(* IEC 61131-3 sources: SRCI/RobotLibrary/Library/POUs/General/MC_RobotTask (part 3) *)

           // Create log entry
           CreateLogMessagePara3 ( Timestamp   := SystemTime,
                                   MessageType := MessageType.CMD,
                                   Severity    := Severity.DEBUG,
                                   MessageCode := 0,
                                   MessageText := 'SyncLoadData: Synchronization of Load[{1}] triggered by PLC, SyncMode = {2}, SyncTime = {3}, SyncDirection = PLC -> RC',
                                   Para1       :=  DINT_TO_STRING(_rSyncIdx),
                                   Para2       :=  SYNC_MODE_TO_STRING(AxesGroup.Parameter.Plc.Parameter.SynchronizationModes.Load[SyncTime.AFTER_START_UP]),
                                   Para3       :=  SYNC_TIME_TO_STRING(SyncTime.AFTER_START_UP));
                                   RETURN;
         END_IF

         // Conflict triggered by RC ?
         IF ( NOT AxesGroup.State.SyncStateRc.InSync.Load )
         THEN
           // get changed index
          _rSyncIdx := LIMIT(1, AxesGroup.State.SyncStateRc.UnSyncNo.Load, AxesGroup.State.UnifiedLoadIndex); //  !!! Attention : 0 is not allowed - LoadData starts with 1 !!!
           // set timeout
           SetTimeout(PT := _rTimeout, rTimer := _rTimer);
           // inc step counter
          _rStep := 20; // -> read RC data an write it to PLC

           // Create log entry
           CreateLogMessagePara3 ( Timestamp   := SystemTime,
                                   MessageType := MessageType.CMD,
                                   Severity    := Severity.DEBUG,
                                   MessageCode := 0,
                                   MessageText := 'SyncLoadData: Synchronization of Load[{1}] triggered by RC, SyncMode = {2}, SyncTime = {3}, SyncDirection = RC -> PLC',
                                   Para1       :=  DINT_TO_STRING(_rSyncIdx),
                                   Para2       :=  SYNC_MODE_TO_STRING(AxesGroup.Parameter.Plc.Parameter.SynchronizationModes.Load[SyncTime.AFTER_START_UP]),
                                   Para3       :=  SYNC_TIME_TO_STRING(SyncTime.AFTER_START_UP));
                                   RETURN;
  			 END_IF

         // set timeout
         SetTimeout(PT := _rTimeout, rTimer := _rTimer);
         // jump back
        //_rStep := 10;

    // ------------------------------------------
    // Read Data from RC and write it to PLC
    // ------------------------------------------
    20 : IF (( NOT _readLoadData.Busy  ) AND
             ( NOT _readLoadData.Error ))
         THEN
           // set command parameter
          _readLoadData.ParCmd.LoadNo := _rSyncIdx;
           // execute command
          _readLoadData.Execute := TRUE;
           // set timeout
           SetTimeout(PT := _rTimeout, rTimer := _rTimer);
           // inc step counter
          _rStep := _rStep + 1;
         ELSE
           // check error ?
           IF (_readLoadData.Error)
           THEN
             ErrorID     := _readLoadData.ErrorID;
             ErrorAddTxt := _readLoadData.ErrorAddTxt;
           END_IF

           // timeout exceeded ?
           IF (CheckTimeout(_rTimer) = RobotLibraryConstants.OK)
           THEN
             ErrorID     := RobotLibraryErrorIdEnum.ERR_TIMEOUT_CMD;
             ErrorAddTxt := CONCAT(_stepName, DINT_TO_STRING(_rStep));
           END_IF
         END_IF

    21 : IF (( NOT _readLoadData.Busy  ) AND
             ( NOT _readLoadData.Error ) AND
             (     _readLoadData.Done  ))
         THEN
           // reset execution
          _readLoadData.Execute := FALSE;
           // update internal Load data
           LoadData[_rSyncIdx].Data := _readLoadData.OutCmd.LoadData;
          _loadData[_rSyncIdx].Data := _readLoadData.OutCmd.LoadData;
           // set available bit
           LoadData[_rSyncIdx].Available := TRUE;
          _loadData[_rSyncIdx].Available := TRUE;
           // set timeout
           SetTimeout(PT := _rTimeout, rTimer := _rTimer);
           // inc step counter
          _rStep := 10; // -> jump to after startup
         ELSE
           // check error ?
           IF (_readLoadData.Error)
           THEN
             ErrorID     := _readLoadData.ErrorID;
             ErrorAddTxt := _readLoadData.ErrorAddTxt;
             // reset available bit
             LoadData[_rSyncIdx].Available := FALSE;
            _loadData[_rSyncIdx].Available := FALSE;
           END_IF

           // timeout exceeded ?
           IF (CheckTimeout(_rTimer) = RobotLibraryConstants.OK)
           THEN
             ErrorID     := RobotLibraryErrorIdEnum.ERR_TIMEOUT_CMD;
             ErrorAddTxt := CONCAT(_stepName, DINT_TO_STRING(_rStep));
           END_IF
         END_IF

    // ------------------------------------------
    // Write data from PLC to RC
    // ------------------------------------------
    30 : IF (( NOT _writeLoadData.Busy  ) AND
             ( NOT _writeLoadData.Error ))
         THEN
           // set command parameter
          _writeLoadData.ParCmd.LoadNo   := _rSyncIdx;
          _writeLoadData.ParCmd.LoadData :=  LoadData[_rSyncIdx].Data;
           // execute command
          _writeLoadData.Execute := TRUE;
           // set timeout
           SetTimeout(PT := _rTimeout, rTimer := _rTimer);
           // inc step counter
          _rStep := _rStep + 1;
         ELSE
           // check error ?
           IF (_writeLoadData.Error)
           THEN
             ErrorID     := _writeLoadData.ErrorID;
             ErrorAddTxt := _writeLoadData.ErrorAddTxt;;
           END_IF

           // timeout exceeded ?
           IF (CheckTimeout(_rTimer) = RobotLibraryConstants.OK)
           THEN
             ErrorID     := RobotLibraryErrorIdEnum.ERR_TIMEOUT_CMD;
             ErrorAddTxt := CONCAT(_stepName, DINT_TO_STRING(_rStep));
           END_IF
         END_IF

    31 : IF (( NOT _writeLoadData.Busy  ) AND
             ( NOT _writeLoadData.Error ) AND
             (     _writeLoadData.Done  ))
         THEN
           // execute command
          _writeLoadData.Execute := FALSE;
           // update internal Load data
          _loadData[_rSyncIdx] := LoadData[_rSyncIdx];
           // set available bit
           LoadData[_rSyncIdx].Available := TRUE;
          _loadData[_rSyncIdx].Available := TRUE;
           // set timeout
           SetTimeout(PT := _rTimeout, rTimer := _rTimer);
           // inc step counter
          _rStep := 10; // -> jump to after startup;
         ELSE
           // check error ?
           IF (_writeLoadData.Error)
           THEN
             WarningID := RobotLibraryWarningIdEnum.WARN_LOAD_SYNC_FAILED_BY_ERROR_OF_READ_OR_WRITE_CMD;
             // reset available bit
             LoadData[_rSyncIdx].Available := FALSE;
            _loadData[_rSyncIdx].Available := FALSE;
           END_IF

           // timeout exceeded ?
           IF (CheckTimeout(_rTimer) = RobotLibraryConstants.OK)
           THEN
             ErrorID     := RobotLibraryErrorIdEnum.ERR_TIMEOUT_CMD;
             ErrorAddTxt := CONCAT(_stepName, DINT_TO_STRING(_rStep));
           END_IF
         END_IF

  ELSE
    // invalid step
    ErrorID     := RobotLibraryErrorIdEnum.ERR_INVALID_STEP;
    ErrorAddTxt := CONCAT(_stepName , DINT_TO_STRING(_stepCmd));
  END_CASE

END_METHOD

METHOD PRIVATE HandleSyncRobotDefaultDynamics
VAR_IN_OUT
   /// Robot assignment of function
  AxesGroup       : AxesGroup;
  /// Default dynamics stored on PLC. For more information refer to 5.5.7
  DefaultDynamics : DefaultDynamics;
END_VAR

VAR
  /// Internal step counter name
 _stepName        : STRING;
  /// Internal reference to step counter
 _rStep           : REFERENCE TO DINT;
  /// Internal reference to timer
 _rTimer          : REFERENCE TO TON;
  /// Internal reference to timeout
 _rTimeout        : REFERENCE TO TIME;
  /// Internal reference to synchroniztion index
 _rSyncIdx        : REFERENCE TO USINT;
  /// internal bit for condition found
 _found           : BOOL;
  /// empty data set to reset all DataChanged bits
 _dataChangedNone : AxesGroupStateDataChanged;
END_VAR

  // Set internal references
  _stepName      :=   '_stepSyncDefaultDynamics = ';
  _rStep       REF=    _stepSyncDefaultDynamics;
  _rTimer      REF=   _timerSyncDefaultDynamics;
  _rTimeout    REF= _timeoutSyncDefaultDynamics;

  CASE _rStep
  OF
    0: // Check initialisation configured ?
       IF (( _parCfg.PLC.Parameter.SynchronizationModes.DefaultDynamics[SyncTime.DURING_START_UP] = SyncMode.NO_SYNCHRONIZATION ) AND
           ( _parCfg.PLC.Parameter.SynchronizationModes.DefaultDynamics[SyncTime. AFTER_START_UP] = SyncMode.NO_SYNCHRONIZATION ))
       THEN
         RETURN;
       END_IF

       // wait for initialisation done
       IF  ((     AxesGroup.State.RobotData.RCSupportedFunctions .ReadRobotDefaultDynamics ) AND
            (     AxesGroup.State.RobotData.RCSupportedFunctions.WriteRobotDefaultDynamics ) AND
            (     AxesGroup.State.Initialized                                              ) AND
            ( NOT Error                                                                    ))
       THEN
         // Create log entry
         CreateLogMessagePara1 ( Timestamp   := SystemTime,
                                 MessageType := MessageType.CMD,
                                 Severity    := Severity.DEBUG,
                                 MessageCode := 0,
                                 MessageText := 'SyncDefaultDynamics: Start initial reading of DefaultDynamics from RC',
                                 Para1       :=  '');

         // set timeout
         SetTimeout(PT := _rTimeout, rTimer := _rTimer);
         // inc step counter
        _rStep := _rStep + 1;
       END_IF

       // Start read DefaultDynamics
    1: IF (( NOT _readRobotDefaultDynamics .Busy  ) AND
           ( NOT _readRobotDefaultDynamics.Error ))
       THEN
         // execute command
        _readRobotDefaultDynamics.Execute := TRUE;
         // set timeout
         SetTimeout(PT := _rTimeout, rTimer := _rTimer);
         // inc step counter
        _rStep := _rStep + 1;
       ELSE
         // check error ?
         IF ( _readRobotDefaultDynamics.Error ) AND ( WarningID = RobotLibraryWarningIdEnum.NO_WARNING )
         THEN
           WarningID := RobotLibraryWarningIdEnum.WARN_DEFAULT_DYNAMICS_SYNC_FAILED_BY_ERROR_OF_READ_OR_WRITE_CMD;
         END_IF

         // timeout exceeded ?
         IF (CheckTimeout(_rTimer) = RobotLibraryConstants.OK)
         THEN
           ErrorID     := RobotLibraryErrorIdEnum.ERR_TIMEOUT_CMD;
           ErrorAddTxt := CONCAT(_stepName, DINT_TO_STRING(_rStep));
         END_IF
       END_IF

       // Wait DefaultDynamics read
    2: IF (( NOT _readRobotDefaultDynamics.Busy  ) AND
           ( NOT _readRobotDefaultDynamics.Error ) AND
           (     _readRobotDefaultDynamics.Done  ))
       THEN
         // reset execution
        _readRobotDefaultDynamics.Execute := FALSE;
         // Copy data
        _defaultDynamics := _readRobotDefaultDynamics.OutCmd.DynamicValues;
         // Set plc in sync flag
         AxesGroup.State.SyncStatePlc.InSync.DefaultDynamics := TRUE;

         // Check DefaultDynamics data is equal ?
         IF ( NOT IsDefaultDynamicsEqual( Data1 := _defaultDynamics, Data2 := DefaultDynamics, IgnoreTimestamp := TRUE))
         THEN
           // Reset plc in sync flag
           AxesGroup.State.SyncStatePlc.InSync.DefaultDynamics := FALSE;
           // Set data changed flag
           AxesGroup.State.DataChanged.DefaultDynamics := TRUE;
           // set timeout
           SetTimeout(PT := _rTimeout, rTimer := _rTimer);
           // inc step counter
          _rStep := _rStep + 1;

           // Create log entry
           CreateLogMessagePara1 ( Timestamp   := SystemTime,
                                   MessageType := MessageType.CMD,
                                   Severity    := Severity.DEBUG,
                                   MessageCode := 0,
                                   MessageText := 'SyncDefaultDynamics: Detected a difference in DefaultDynamics between PLC and RC',
                                   Para1       :=  '');

           // Check synchronisation is enabled ?
           IF ( NOT  AxesGroup.State.DataEnableSync.EnableSyncDefaultDynamics ) AND (InfoID = RobotLibraryInfoIdEnum.NO_INFO )
           THEN
             InfoID := RobotLibraryInfoIdEnum.INFO_SYNC_DEFAULT_DYNAMICS_DISABLED;
  				 END_IF

           // Check user interaction needed ?
           IF ( AxesGroup.Parameter.Plc.Parameter.SyncUserInteraction.DefaultDynamics ) AND ( WarningID = RobotLibraryWarningIdEnum.NO_WARNING )
           THEN
             WarningID := RobotLibraryWarningIdEnum.WARN_DEFAULT_DYNAMICS_SYNC_ERROR;
  				 END_IF
  			 END_IF
       ELSE
         // check error ?
         IF (_readRobotDefaultDynamics.Error)
         THEN
           // Set warning
           WarningID := RobotLibraryWarningIdEnum.WARN_DEFAULT_DYNAMICS_SYNC_FAILED_BY_ERROR_OF_READ_OR_WRITE_CMD;
         END_IF

         // timeout exceeded ?
         IF (CheckTimeout(_rTimer) = RobotLibraryConstants.OK)
         THEN
           ErrorID     := RobotLibraryErrorIdEnum.ERR_TIMEOUT_CMD;
           ErrorAddTxt := CONCAT(_stepName, DINT_TO_STRING(_rStep));
         END_IF
       END_IF

       // Check synchronisation state ?
    3: IF ((  NOT AxesGroup.State.DataChanged.DefaultDynamics                                                                                    ) OR
           (      AxesGroup.Parameter.Plc.Parameter.SynchronizationModes.DefaultDynamics[SyncTime.DURING_START_UP] = SyncMode.NO_SYNCHRONIZATION ))
       THEN
         // Update bit for data in sync
         AxesGroup.State.SyncStatePlc.InSync.DefaultDynamics := NOT AxesGroup.State.DataChanged.DefaultDynamics ;
         // set timeout
         SetTimeout(PT := _rTimeout, rTimer := _rTimer);
         // inc step counter
        _rStep := 10; // -> jump to after startup

         // Create log entry
         CreateLogMessagePara1 ( Timestamp   := SystemTime,
                                 MessageType := MessageType.CMD,
                                 Severity    := Severity.DEBUG,
                                 MessageCode := 0,
                                 MessageText := 'SyncDefaultDynamics: Synchronization Startup Phase done',
                                 Para1       :=  '' );
       ELSE
         // Check user interaction needed ?
         IF ( NOT AxesGroup.Parameter.Plc.Parameter.SyncUserInteraction.DefaultDynamics )
         THEN
           CASE AxesGroup.Parameter.Plc.Parameter.SynchronizationModes.DefaultDynamics[SyncTime.DURING_START_UP] OF

             SyncMode.SERVER_TO_CLIENT :

               // Overwrite PLC data with RC data
               DefaultDynamics := _defaultDynamics;
               // Reset data changed flags
               AxesGroup.State.DataChanged.DefaultDynamics := _dataChangedNone.DefaultDynamics;
               // Reset Synchronizing flag
               AxesGroup.State.Synchronizing.DefaultDynamics := FALSE;
               // Set plc in sync flag
               AxesGroup.State.SyncStatePlc.InSync.DefaultDynamics := TRUE;
               // set timeout
               SetTimeout(PT := _rTimeout, rTimer := _rTimer);
               // inc step counter
              _rStep := 10; // -> jump to after startup

              // Create log entry
              CreateLogMessagePara2 ( Timestamp   := SystemTime,
                                      MessageType := MessageType.CMD,
                                      Severity    := Severity.DEBUG,
                                      MessageCode := 0,
                                      MessageText := 'SyncDefaultDynamics: Synchronization of DefaultDynamics triggered by StartUp-Compare, SyncMode = {1}, SyncTime = {2}, SyncDirection = RC -> PLC',
                                      Para1       :=  SYNC_MODE_TO_STRING(AxesGroup.Parameter.Plc.Parameter.SynchronizationModes.DefaultDynamics[SyncTime.DURING_START_UP]),
                                      Para2       :=  SYNC_TIME_TO_STRING(SyncTime.DURING_START_UP));
              // Create log entry
              CreateLogMessagePara1 ( Timestamp   := SystemTime,
                                      MessageType := MessageType.CMD,
                                      Severity    := Severity.DEBUG,
                                      MessageCode := 0,
                                      MessageText := 'SyncDefaultDynamics: Applied the initial read DefaultDynamics from RC',
                                      Para1       :=  '' );

  				   SyncMode.CLIENT_TO_SERVER : ;

               IF ( AxesGroup.State.DataChanged.DefaultDynamics )
               THEN
                 // Reset plc in sync flag
                 AxesGroup.State.SyncStatePlc.InSync.DefaultDynamics := FALSE;
                 // Set Synchronizing flag
                 AxesGroup.State.Synchronizing.DefaultDynamics := TRUE;
                 // set timeout
                 SetTimeout(PT := _rTimeout, rTimer := _rTimer);
                 // inc step counter
                _rStep := _rStep +1; // -> write PLC data to RC
                 // Create log entry
                 CreateLogMessagePara2 ( Timestamp   := SystemTime,
                                         MessageType := MessageType.CMD,
                                         Severity    := Severity.DEBUG,
                                         MessageCode := 0,
                                         MessageText := 'SyncDefaultDynamics: Synchronization of DefaultDynamics triggered by StartUp-Compare, SyncMode = {1}, SyncTime = {2}, SyncDirection = PLC -> RC',
                                         Para1       :=  SYNC_MODE_TO_STRING(AxesGroup.Parameter.Plc.Parameter.SynchronizationModes.DefaultDynamics[SyncTime.DURING_START_UP]),
                                         Para2       :=  SYNC_TIME_TO_STRING(SyncTime.DURING_START_UP));
               ELSE
                 // Reset data changed flags
                 AxesGroup.State.DataChanged.DefaultDynamics := _dataChangedNone.DefaultDynamics;
                 // Reset Synchronizing flag
                 AxesGroup.State.Synchronizing.DefaultDynamics := FALSE;
                 // Set plc in sync flag
                 AxesGroup.State.SyncStatePlc.InSync.DefaultDynamics := TRUE;
                 // set timeout
                 SetTimeout(PT := _rTimeout, rTimer := _rTimer);
                 // inc step counter
                _rStep := 10; // -> jump to after startup
  				     END_IF
           ELSE
             // invalid sync mode for startup
             ErrorID := RobotLibraryErrorIdEnum.ERR_SYNC_MODE_INVALID;
   	       END_CASE
         END_IF
       END_IF

       // Start write DefaultDynamics data
    4: IF (( NOT _writeRobotDefaultDynamics.Busy  ) AND
           ( NOT _writeRobotDefaultDynamics.Error ))
       THEN
         // set command parameter
        _writeRobotDefaultDynamics.ParCmd.DynamicValues :=  DefaultDynamics;
         // execute command
        _writeRobotDefaultDynamics.Execute := TRUE;
         // set timeout
         SetTimeout(PT := _rTimeout, rTimer := _rTimer);
         // inc step counter
        _rStep := _rStep + 1;
       ELSE
         // check error ?
         IF (_writeRobotDefaultDynamics.Error)
         THEN
           ErrorID     := _writeRobotDefaultDynamics.ErrorID;
           ErrorAddTxt := _writeRobotDefaultDynamics.ErrorAddTxt;;
         END_IF

         // timeout exceeded ?
         IF (CheckTimeout(_rTimer) = RobotLibraryConstants.OK)
         THEN
           ErrorID     := RobotLibraryErrorIdEnum.ERR_TIMEOUT_CMD;
           ErrorAddTxt := CONCAT(_stepName, DINT_TO_STRING(_rStep));
         END_IF
       END_IF

       // Wait DefaultDynamics data written ?
    5: IF (( NOT _writeRobotDefaultDynamics.Busy  ) AND
           ( NOT _writeRobotDefaultDynamics.Error ) AND
           (     _writeRobotDefaultDynamics.Done  ))
       THEN
         // execute command
        _writeRobotDefaultDynamics.Execute := FALSE;
         // apply DefaultDynamics data to internal DefaultDynamics data
        _defaultDynamics := DefaultDynamics;
         // reset data changed bit
         AxesGroup.State.DataChanged.DefaultDynamics := FALSE;
         // set timeout
         SetTimeout(PT := _rTimeout, rTimer := _rTimer);
         // dec step counter
        _rStep := _rStep - 2;
       ELSE
         // check error ?
         IF (_writeRobotDefaultDynamics.Error)
         THEN
           WarningID := RobotLibraryWarningIdEnum.WARN_DEFAULT_DYNAMICS_SYNC_FAILED_BY_ERROR_OF_READ_OR_WRITE_CMD;
         END_IF

         // timeout exceeded ?
         IF (CheckTimeout(_rTimer) = RobotLibraryConstants.OK)
         THEN
           ErrorID     := RobotLibraryErrorIdEnum.ERR_TIMEOUT_CMD;
           ErrorAddTxt := CONCAT(_stepName, DINT_TO_STRING(_rStep));
         END_IF
       END_IF

    // --------------------------------------------
    // SyncMode after startup :
    // --------------------------------------------

    10 :// check synchronisation active ?
         IF ( AxesGroup.Parameter.Plc.Parameter.SynchronizationModes.DefaultDynamics[SyncTime.AFTER_START_UP] = SyncMode.NO_SYNCHRONIZATION)
         THEN
           RETURN;
         END_IF

         // compare DefaultDynamics data
         AxesGroup.State.DataChanged.DefaultDynamics := NOT IsDefaultDynamicsEqual( Data1 := DefaultDynamics, Data2 := _defaultDynamics, IgnoreTimestamp := FALSE);

         // Check DefaultDynamics data changed ?
         IF (AxesGroup.State.DataChanged.DefaultDynamics)
         THEN
           // Create log entry
           CreateLogMessagePara1 ( Timestamp   := SystemTime,
                                   MessageType := MessageType.CMD,
                                   Severity    := Severity.DEBUG,
                                   MessageCode := 0,
                                   MessageText := 'SyncDefaultDynamics: Detected a local change of DefaultDynamics on PLC, SyncTime = {1}',
                                   Para1       :=  SYNC_TIME_TO_STRING(SyncTime.AFTER_START_UP));
         END_IF

         // Update plc in sync flag
         AxesGroup.State.SyncStatePlc.InSync.DefaultDynamics := NOT AxesGroup.State.DataChanged.DefaultDynamics;

         // Check synchronization is needed ?
         IF ( NOT AxesGroup.State.SyncStatePlc.InSync.DefaultDynamics ) XOR
            ( NOT AxesGroup.State.SyncStateRc .InSync.DefaultDynamics )
         THEN
           CASE AxesGroup.Parameter.Plc.Parameter.SynchronizationModes.DefaultDynamics[SyncTime.AFTER_START_UP]
           OF
             // NO_SYNCHRONIZATION
             SyncMode.NO_SYNCHRONIZATION : ; // no further action

             // CLIENT_TO_SERVER
             SyncMode.CLIENT_TO_SERVER :
               // set timeout
               SetTimeout(PT := _rTimeout, rTimer := _rTimer);
               // inc step counter
              _rStep := 11;

             // SERVER_TO_CLIENT
             SyncMode.SERVER_TO_CLIENT :
               // set timeout
               SetTimeout(PT := _rTimeout, rTimer := _rTimer);
               // inc step counter
              _rStep := 12;

             // AUTOMATIC
             SyncMode.AUTOMATIC :
               // set timeout
               SetTimeout(PT := _rTimeout, rTimer := _rTimer);
               // inc step counter
              _rStep := 13;
           END_CASE
         ELSE
           // datas changeḍ on both sides ? -> Warning
           IF (( NOT AxesGroup.State.SyncStatePlc.InSync.DefaultDynamics ) AND
               ( NOT AxesGroup.State.SyncStateRc .InSync.DefaultDynamics ))
           THEN
             WarningID := RobotLibraryWarningIdEnum.WARN_DEFAULT_DYNAMICS_SYNC_BOTH_SIDES_CHANGED;
           END_IF
         END_IF

    // ------------------------------------------
    // SyncMode : CLIENT_TO_SERVER
    // ------------------------------------------
    11 : // Conflict triggerd by PLC ?
         IF ( NOT AxesGroup.State.SyncStatePlc.InSync.DefaultDynamics )
         THEN
           // set timeout
           SetTimeout(PT := _rTimeout, rTimer := _rTimer);
           // inc step counter
          _rStep := 30; // -> write PLC data to RC

           // Create log entry
           CreateLogMessagePara2 ( Timestamp   := SystemTime,
                                   MessageType := MessageType.CMD,
                                   Severity    := Severity.DEBUG,
                                   MessageCode := 0,
                                   MessageText := 'SyncDefaultDynamics: Synchronization of DefaultDynamics triggered by PLC, SyncMode = {1}, SyncTime = {2}, SyncDirection = PLC -> RC',
                                   Para1       :=  SYNC_MODE_TO_STRING(AxesGroup.Parameter.Plc.Parameter.SynchronizationModes.DefaultDynamics[SyncTime.AFTER_START_UP]),
                                   Para2       :=  SYNC_TIME_TO_STRING(SyncTime.AFTER_START_UP));
                                   RETURN;
         END_IF

         // Conflict triggered by RC ?
         IF ( NOT AxesGroup.State.SyncStateRc.InSync.DefaultDynamics )
         THEN
           // set timeout
           SetTimeout(PT := _rTimeout, rTimer := _rTimer);
           // inc step counter
          _rStep := 30; // -> write PLC data to RC

           // Create log entry
           CreateLogMessagePara2 ( Timestamp   := SystemTime,
                                   MessageType := MessageType.CMD,
                                   Severity    := Severity.DEBUG,
                                   MessageCode := 0,
                                   MessageText := 'SyncDefaultDynamics: Synchronization of DefaultDynamics triggered by RC, SyncMode = {1}, SyncTime = {2}, SyncDirection = PLC -> RC',
                                   Para1       :=  SYNC_MODE_TO_STRING(AxesGroup.Parameter.Plc.Parameter.SynchronizationModes.DefaultDynamics[SyncTime.AFTER_START_UP]),
                                   Para2       :=  SYNC_TIME_TO_STRING(SyncTime.AFTER_START_UP));
                                   RETURN;
  			 END_IF

         // set timeout
         SetTimeout(PT := _rTimeout, rTimer := _rTimer);
         // jump back
        _rStep := 10;

    // ------------------------------------------
    // SyncMode : SERVER_TO_CLIENT
    // ------------------------------------------
    12 : // Conflict triggerd by PLC ?
         IF ( NOT AxesGroup.State.SyncStatePlc.InSync.DefaultDynamics )
         THEN
           // set timeout
           SetTimeout(PT := _rTimeout, rTimer := _rTimer);
           // inc step counter
          _rStep := 20; // -> read RC data and write it to PLC

           // Create log entry
           CreateLogMessagePara2 ( Timestamp   := SystemTime,
                                   MessageType := MessageType.CMD,
                                   Severity    := Severity.DEBUG,
                                   MessageCode := 0,
                                   MessageText := 'SyncDefaultDynamics: Synchronization of DefaultDynamics triggered by PLC, SyncMode = {1}, SyncTime = {2}, SyncDirection = RC -> PLC',
                                   Para1       :=  SYNC_MODE_TO_STRING(AxesGroup.Parameter.Plc.Parameter.SynchronizationModes.DefaultDynamics[SyncTime.AFTER_START_UP]),
                                   Para2       :=  SYNC_TIME_TO_STRING(SyncTime.AFTER_START_UP));
                                   RETURN;
         END_IF

         // Conflict triggered by RC ?
         IF ( NOT AxesGroup.State.SyncStateRc.InSync.DefaultDynamics )
         THEN
           // set timeout
           SetTimeout(PT := _rTimeout, rTimer := _rTimer);
           // inc step counter
          _rStep := 20; // -> read RC data and write it to PLC

           // Create log entry
           CreateLogMessagePara2 ( Timestamp   := SystemTime,
                                   MessageType := MessageType.CMD,
                                   Severity    := Severity.DEBUG,
                                   MessageCode := 0,
                                   MessageText := 'SyncDefaultDynamics: Synchronization of DefaultDynamics triggered by RC, SyncMode = {1}, SyncTime = {2}, SyncDirection = RC -> PLC',
                                   Para1       :=  SYNC_MODE_TO_STRING(AxesGroup.Parameter.Plc.Parameter.SynchronizationModes.DefaultDynamics[SyncTime.AFTER_START_UP]),
                                   Para2       :=  SYNC_TIME_TO_STRING(SyncTime.AFTER_START_UP));
                                   RETURN;
  			 END_IF

         // set timeout
         SetTimeout(PT := _rTimeout, rTimer := _rTimer);
         // jump back
        _rStep := 10;

    // ------------------------------------------
    // SyncMode : AUTOMATIC
    // ------------------------------------------
    13 : // Conflict triggerd by PLC ?
         IF ( NOT AxesGroup.State.SyncStatePlc.InSync.DefaultDynamics )
         THEN
           // set timeout
           SetTimeout(PT := _rTimeout, rTimer := _rTimer);
           // inc step counter
          _rStep := 30; // -> write PLC data to RC

           // Create log entry
           CreateLogMessagePara2 ( Timestamp   := SystemTime,
                                   MessageType := MessageType.CMD,
                                   Severity    := Severity.DEBUG,
                                   MessageCode := 0,
                                   MessageText := 'SyncDefaultDynamics: Synchronization of DefaultDynamics triggered by PLC, SyncMode = {1}, SyncTime = {2}, SyncDirection = PLC -> RC',
                                   Para1       :=  SYNC_MODE_TO_STRING(AxesGroup.Parameter.Plc.Parameter.SynchronizationModes.DefaultDynamics[SyncTime.AFTER_START_UP]),
                                   Para2       :=  SYNC_TIME_TO_STRING(SyncTime.AFTER_START_UP));
                                   RETURN;
         END_IF

         // Conflict triggered by RC ?
         IF ( NOT AxesGroup.State.SyncStateRc.InSync.DefaultDynamics )
         THEN
           // set timeout
           SetTimeout(PT := _rTimeout, rTimer := _rTimer);
           // inc step counter
          _rStep := 20; // -> read RC data an write it to PLC

           // Create log entry
           CreateLogMessagePara2 ( Timestamp   := SystemTime,
                                   MessageType := MessageType.CMD,
                                   Severity    := Severity.DEBUG,
                                   MessageCode := 0,
                                   MessageText := 'SyncDefaultDynamics: Synchronization of DefaultDynamics triggered by RC, SyncMode = {1}, SyncTime = {2}, SyncDirection = RC -> PLC',
                                   Para1       :=  SYNC_MODE_TO_STRING(AxesGroup.Parameter.Plc.Parameter.SynchronizationModes.DefaultDynamics[SyncTime.AFTER_START_UP]),
                                   Para2       :=  SYNC_TIME_TO_STRING(SyncTime.AFTER_START_UP));
                                   RETURN;
  			 END_IF

         // set timeout
         SetTimeout(PT := _rTimeout, rTimer := _rTimer);
         // jump back
        //_rStep := 10;

    // ------------------------------------------
    // Read Data from RC and write it to PLC
    // ------------------------------------------
    20 : IF (( NOT _readRobotDefaultDynamics.Busy  ) AND
             ( NOT _readRobotDefaultDynamics.Error ))
         THEN
           // execute command
          _readRobotDefaultDynamics.Execute := TRUE;
           // set timeout
           SetTimeout(PT := _rTimeout, rTimer := _rTimer);
           // inc step counter
          _rStep := _rStep + 1;
         ELSE
           // check error ?
           IF (_readRobotDefaultDynamics.Error)
           THEN
             ErrorID     := _readRobotDefaultDynamics.ErrorID;
             ErrorAddTxt := _readRobotDefaultDynamics.ErrorAddTxt;
           END_IF

           // timeout exceeded ?
           IF (CheckTimeout(_rTimer) = RobotLibraryConstants.OK)
           THEN
             ErrorID     := RobotLibraryErrorIdEnum.ERR_TIMEOUT_CMD;
             ErrorAddTxt := CONCAT(_stepName, DINT_TO_STRING(_rStep));
           END_IF
         END_IF

    21 : IF (( NOT _readRobotDefaultDynamics.Busy  ) AND
             ( NOT _readRobotDefaultDynamics.Error ) AND
             (     _readRobotDefaultDynamics.Done  ))
         THEN
           // reset execution
          _readRobotDefaultDynamics.Execute := FALSE;
           // update internal DefaultDynamics data
           DefaultDynamics := _readRobotDefaultDynamics.OutCmd.DynamicValues;
          _defaultDynamics := _readRobotDefaultDynamics.OutCmd.DynamicValues;
           // set timeout
           SetTimeout(PT := _rTimeout, rTimer := _rTimer);
           // inc step counter
          _rStep := 10; // -> jump to after startup
         ELSE
           // check error ?
           IF (_readRobotDefaultDynamics.Error)
           THEN
             ErrorID     := _readRobotDefaultDynamics.ErrorID;
             ErrorAddTxt := _readRobotDefaultDynamics.ErrorAddTxt;
           END_IF

           // timeout exceeded ?
           IF (CheckTimeout(_rTimer) = RobotLibraryConstants.OK)
           THEN
             ErrorID     := RobotLibraryErrorIdEnum.ERR_TIMEOUT_CMD;
             ErrorAddTxt := CONCAT(_stepName, DINT_TO_STRING(_rStep));
           END_IF
         END_IF

    // ------------------------------------------
    // Write data from PLC to RC
    // ------------------------------------------
    30 : IF (( NOT _writeRobotDefaultDynamics.Busy  ) AND
             ( NOT _writeRobotDefaultDynamics.Error ))
         THEN
           // set command parameter
          _writeRobotDefaultDynamics.ParCmd.DynamicValues :=  DefaultDynamics;
           // execute command
          _writeRobotDefaultDynamics.Execute := TRUE;
           // set timeout
           SetTimeout(PT := _rTimeout, rTimer := _rTimer);
           // inc step counter
          _rStep := _rStep + 1;
         ELSE
           // check error ?
           IF (_writeRobotDefaultDynamics.Error)
           THEN
             ErrorID     := _writeRobotDefaultDynamics.ErrorID;
             ErrorAddTxt := _writeRobotDefaultDynamics.ErrorAddTxt;;
           END_IF

           // timeout exceeded ?
           IF (CheckTimeout(_rTimer) = RobotLibraryConstants.OK)
           THEN
             ErrorID     := RobotLibraryErrorIdEnum.ERR_TIMEOUT_CMD;
             ErrorAddTxt := CONCAT(_stepName, DINT_TO_STRING(_rStep));
           END_IF
         END_IF

    31 : IF (( NOT _writeRobotDefaultDynamics.Busy  ) AND
             ( NOT _writeRobotDefaultDynamics.Error ) AND
             (     _writeRobotDefaultDynamics.Done  ))
         THEN
           // execute command
          _writeRobotDefaultDynamics.Execute := FALSE;
           // update internal DefaultDynamics data
          _defaultDynamics := DefaultDynamics;
           // set timeout
           SetTimeout(PT := _rTimeout, rTimer := _rTimer);
           // inc step counter
          _rStep := 10; // -> jump to after startup;
         ELSE
           // check error ?
           IF (_writeRobotDefaultDynamics.Error)
           THEN
             WarningID := RobotLibraryWarningIdEnum.WARN_DEFAULT_DYNAMICS_SYNC_FAILED_BY_ERROR_OF_READ_OR_WRITE_CMD;
           END_IF

           // timeout exceeded ?
           IF (CheckTimeout(_rTimer) = RobotLibraryConstants.OK)
           THEN
             ErrorID     := RobotLibraryErrorIdEnum.ERR_TIMEOUT_CMD;
             ErrorAddTxt := CONCAT(_stepName, DINT_TO_STRING(_rStep));
           END_IF
         END_IF

  ELSE
    // invalid step
    ErrorID     := RobotLibraryErrorIdEnum.ERR_INVALID_STEP;
    ErrorAddTxt := CONCAT(_stepName , DINT_TO_STRING(_stepCmd));
  END_CASE

END_METHOD

METHOD PRIVATE HandleSyncRobotReferenceDynamics
VAR_IN_OUT
   /// Robot assignment of function
  AxesGroup         : AxesGroup;
  /// Reference dynamics stored on PLC. For more information refer to 5.5.7
  ReferenceDynamics : ReferenceDynamics;
END_VAR

VAR
  /// Internal step counter name
 _stepName        : STRING;
  /// Internal reference to step counter
 _rStep           : REFERENCE TO DINT;
  /// Internal reference to timer
 _rTimer          : REFERENCE TO TON;
  /// Internal reference to timeout
 _rTimeout        : REFERENCE TO TIME;
  /// Internal reference to synchroniztion index
 _rSyncIdx        : REFERENCE TO USINT;
  /// internal bit for condition found
 _found           : BOOL;
  /// empty data set to reset all DataChanged bits
 _dataChangedNone : AxesGroupStateDataChanged;
END_VAR

  // Set internal references
  _stepName      :=   '_stepSyncReferenceDynamics = ';
  _rStep       REF=    _stepSyncReferenceDynamics;
  _rTimer      REF=   _timerSyncReferenceDynamics;
  _rTimeout    REF= _timeoutSyncReferenceDynamics;

  CASE _rStep
  OF
    0: // Check initialisation configured ?
       IF (( _parCfg.PLC.Parameter.SynchronizationModes.ReferenceDynamics[SyncTime.DURING_START_UP] = SyncMode.NO_SYNCHRONIZATION ) AND
           ( _parCfg.PLC.Parameter.SynchronizationModes.ReferenceDynamics[SyncTime. AFTER_START_UP] = SyncMode.NO_SYNCHRONIZATION ))
       THEN
         RETURN;
       END_IF

       // wait for initialisation done
       IF  ((     AxesGroup.State.RobotData.RCSupportedFunctions .ReadRobotReferenceDynamics ) AND
            (     AxesGroup.State.RobotData.RCSupportedFunctions.WriteRobotReferenceDynamics ) AND
            (     AxesGroup.State.Initialized                                              ) AND
            ( NOT Error                                                                    ))
       THEN
         // Create log entry
         CreateLogMessagePara1 ( Timestamp   := SystemTime,
                                 MessageType := MessageType.CMD,
                                 Severity    := Severity.DEBUG,
                                 MessageCode := 0,
                                 MessageText := 'SyncReferenceDynamics: Start initial reading of ReferenceDynamics from RC',
                                 Para1       :=  '');

         // set timeout
         SetTimeout(PT := _rTimeout, rTimer := _rTimer);
         // inc step counter
        _rStep := _rStep + 1;
       END_IF

       // Start read ReferenceDynamics
    1: IF (( NOT _readRobotReferenceDynamics .Busy  ) AND
           ( NOT _readRobotReferenceDynamics.Error ))
       THEN
         // execute command
        _readRobotReferenceDynamics.Execute := TRUE;
         // set timeout
         SetTimeout(PT := _rTimeout, rTimer := _rTimer);
         // inc step counter
        _rStep := _rStep + 1;
       ELSE
         // check error ?
         IF ( _readRobotReferenceDynamics.Error ) AND ( WarningID = RobotLibraryWarningIdEnum.NO_WARNING )
         THEN
           WarningID := RobotLibraryWarningIdEnum.WARN_REFERENCE_DYNAMICS_SYNC_FAILED_BY_ERROR_OF_READ_OR_WRITE_CMD;
         END_IF

         // timeout exceeded ?
         IF (CheckTimeout(_rTimer) = RobotLibraryConstants.OK)
         THEN
           ErrorID     := RobotLibraryErrorIdEnum.ERR_TIMEOUT_CMD;
           ErrorAddTxt := CONCAT(_stepName, DINT_TO_STRING(_rStep));
         END_IF
       END_IF

       // Wait ReferenceDynamics read
    2: IF (( NOT _readRobotReferenceDynamics.Busy  ) AND
           ( NOT _readRobotReferenceDynamics.Error ) AND
           (     _readRobotReferenceDynamics.Done  ))
       THEN
         // reset execution
        _readRobotReferenceDynamics.Execute := FALSE;
         // Copy data
        _referenceDynamics := _readRobotReferenceDynamics.OutCmd.DynamicValues;
         // Set plc in sync flag
         AxesGroup.State.SyncStatePlc.InSync.ReferenceDynamics := TRUE;

         // Check ReferenceDynamics data is equal ?
         IF ( NOT IsReferenceDynamicsEqual( Data1 := _referenceDynamics, Data2 := ReferenceDynamics, IgnoreTimestamp := TRUE))
         THEN
           // Reset plc in sync flag
           AxesGroup.State.SyncStatePlc.InSync.ReferenceDynamics := FALSE;
           // Set data changed flag
           AxesGroup.State.DataChanged.ReferenceDynamics := TRUE;
           // set timeout
           SetTimeout(PT := _rTimeout, rTimer := _rTimer);
           // inc step counter
          _rStep := _rStep + 1;

           // Create log entry
           CreateLogMessagePara1 ( Timestamp   := SystemTime,
                                   MessageType := MessageType.CMD,
                                   Severity    := Severity.DEBUG,
                                   MessageCode := 0,
                                   MessageText := 'SyncReferenceDynamics: Detected a difference in ReferenceDynamics between PLC and RC',
                                   Para1       :=  '');

           // Check synchronisation is enabled ?
           IF ( NOT  AxesGroup.State.DataEnableSync.EnableSyncReferenceDynamics ) AND (InfoID = RobotLibraryInfoIdEnum.NO_INFO )
           THEN
             InfoID := RobotLibraryInfoIdEnum.INFO_SYNC_REFERENCE_DYNAMICS_DISABLED;
  				 END_IF

           // Check user interaction needed ?
           IF ( AxesGroup.Parameter.Plc.Parameter.SyncUserInteraction.ReferenceDynamics ) AND ( WarningID = RobotLibraryWarningIdEnum.NO_WARNING )
           THEN
             WarningID := RobotLibraryWarningIdEnum.WARN_REFERENCE_DYNAMICS_SYNC_ERROR;
  				 END_IF
  			 END_IF
       ELSE
         // check error ?
         IF (_readRobotReferenceDynamics.Error)
         THEN
           // Set warning
           WarningID := RobotLibraryWarningIdEnum.WARN_REFERENCE_DYNAMICS_SYNC_FAILED_BY_ERROR_OF_READ_OR_WRITE_CMD;
         END_IF

         // timeout exceeded ?
         IF (CheckTimeout(_rTimer) = RobotLibraryConstants.OK)
         THEN
           ErrorID     := RobotLibraryErrorIdEnum.ERR_TIMEOUT_CMD;
           ErrorAddTxt := CONCAT(_stepName, DINT_TO_STRING(_rStep));
         END_IF
       END_IF

       // Check synchronisation state ?
    3: IF ((  NOT AxesGroup.State.DataChanged.ReferenceDynamics                                                                                    ) OR
           (      AxesGroup.Parameter.Plc.Parameter.SynchronizationModes.ReferenceDynamics[SyncTime.DURING_START_UP] = SyncMode.NO_SYNCHRONIZATION ))
       THEN
         // Update bit for data in sync
         AxesGroup.State.SyncStatePlc.InSync.ReferenceDynamics := NOT AxesGroup.State.DataChanged.ReferenceDynamics ;
         // set timeout
         SetTimeout(PT := _rTimeout, rTimer := _rTimer);
         // inc step counter
        _rStep := 10; // -> jump to after startup

         // Create log entry
         CreateLogMessagePara1 ( Timestamp   := SystemTime,
                                 MessageType := MessageType.CMD,
                                 Severity    := Severity.DEBUG,
                                 MessageCode := 0,
                                 MessageText := 'SyncReferenceDynamics: Synchronization Startup Phase done',
                                 Para1       :=  '' );
       ELSE
         // Check user interaction needed ?
         IF ( NOT AxesGroup.Parameter.Plc.Parameter.SyncUserInteraction.ReferenceDynamics )
         THEN
           CASE AxesGroup.Parameter.Plc.Parameter.SynchronizationModes.ReferenceDynamics[SyncTime.DURING_START_UP] OF

             SyncMode.SERVER_TO_CLIENT :

               // Overwrite PLC data with RC data
               ReferenceDynamics := _referenceDynamics;
               // Reset data changed flags
               AxesGroup.State.DataChanged.ReferenceDynamics := _dataChangedNone.ReferenceDynamics;
               // Reset Synchronizing flag
               AxesGroup.State.Synchronizing.ReferenceDynamics := FALSE;
               // Set plc in sync flag
               AxesGroup.State.SyncStatePlc.InSync.ReferenceDynamics := TRUE;
               // set timeout
               SetTimeout(PT := _rTimeout, rTimer := _rTimer);
               // inc step counter
              _rStep := 10; // -> jump to after startup

              // Create log entry
              CreateLogMessagePara2 ( Timestamp   := SystemTime,
                                      MessageType := MessageType.CMD,
                                      Severity    := Severity.DEBUG,
                                      MessageCode := 0,
                                      MessageText := 'SyncReferenceDynamics: Synchronization of ReferenceDynamics triggered by StartUp-Compare, SyncMode = {1}, SyncTime = {2}, SyncDirection = RC -> PLC',
                                      Para1       :=  SYNC_MODE_TO_STRING(AxesGroup.Parameter.Plc.Parameter.SynchronizationModes.ReferenceDynamics[SyncTime.DURING_START_UP]),
                                      Para2       :=  SYNC_TIME_TO_STRING(SyncTime.DURING_START_UP));
              // Create log entry
              CreateLogMessagePara1 ( Timestamp   := SystemTime,
                                      MessageType := MessageType.CMD,
                                      Severity    := Severity.DEBUG,
                                      MessageCode := 0,
                                      MessageText := 'SyncReferenceDynamics: Applied the initial read ReferenceDynamics from RC',
                                      Para1       :=  '' );

  				   SyncMode.CLIENT_TO_SERVER : ;

               IF ( AxesGroup.State.DataChanged.ReferenceDynamics )
               THEN
                 // Reset plc in sync flag
                 AxesGroup.State.SyncStatePlc.InSync.ReferenceDynamics := FALSE;
                 // Set Synchronizing flag
                 AxesGroup.State.Synchronizing.ReferenceDynamics := TRUE;
                 // set timeout
                 SetTimeout(PT := _rTimeout, rTimer := _rTimer);
                 // inc step counter
                _rStep := _rStep +1; // -> write PLC data to RC
                 // Create log entry
                 CreateLogMessagePara2 ( Timestamp   := SystemTime,
                                         MessageType := MessageType.CMD,
                                         Severity    := Severity.DEBUG,
                                         MessageCode := 0,
                                         MessageText := 'SyncReferenceDynamics: Synchronization of ReferenceDynamics triggered by StartUp-Compare, SyncMode = {1}, SyncTime = {2}, SyncDirection = PLC -> RC',
                                         Para1       :=  SYNC_MODE_TO_STRING(AxesGroup.Parameter.Plc.Parameter.SynchronizationModes.ReferenceDynamics[SyncTime.DURING_START_UP]),
                                         Para2       :=  SYNC_TIME_TO_STRING(SyncTime.DURING_START_UP));
               ELSE
                 // Reset data changed flags
                 AxesGroup.State.DataChanged.ReferenceDynamics := _dataChangedNone.ReferenceDynamics;
                 // Reset Synchronizing flag
                 AxesGroup.State.Synchronizing.ReferenceDynamics := FALSE;
                 // Set plc in sync flag
                 AxesGroup.State.SyncStatePlc.InSync.ReferenceDynamics := TRUE;
                 // set timeout
                 SetTimeout(PT := _rTimeout, rTimer := _rTimer);
                 // inc step counter
                _rStep := 10; // -> jump to after startup
  				     END_IF
           ELSE
             // invalid sync mode for startup
             ErrorID := RobotLibraryErrorIdEnum.ERR_SYNC_MODE_INVALID;
   	       END_CASE
         END_IF
       END_IF

       // Start write ReferenceDynamics data
    4: IF (( NOT _writeRobotReferenceDynamics.Busy  ) AND
           ( NOT _writeRobotReferenceDynamics.Error ))
       THEN
         // set command parameter
        _writeRobotReferenceDynamics.ParCmd.DynamicValues :=  ReferenceDynamics;
         // execute command
        _writeRobotReferenceDynamics.Execute := TRUE;
         // set timeout
         SetTimeout(PT := _rTimeout, rTimer := _rTimer);
         // inc step counter
        _rStep := _rStep + 1;
       ELSE
         // check error ?
         IF (_writeRobotReferenceDynamics.Error)
         THEN
           ErrorID     := _writeRobotReferenceDynamics.ErrorID;
           ErrorAddTxt := _writeRobotReferenceDynamics.ErrorAddTxt;;
         END_IF

         // timeout exceeded ?
         IF (CheckTimeout(_rTimer) = RobotLibraryConstants.OK)
         THEN
           ErrorID     := RobotLibraryErrorIdEnum.ERR_TIMEOUT_CMD;
           ErrorAddTxt := CONCAT(_stepName, DINT_TO_STRING(_rStep));
         END_IF
       END_IF

       // Wait ReferenceDynamics data written ?
    5: IF (( NOT _writeRobotReferenceDynamics.Busy  ) AND
           ( NOT _writeRobotReferenceDynamics.Error ) AND
           (     _writeRobotReferenceDynamics.Done  ))
       THEN
         // execute command
        _writeRobotReferenceDynamics.Execute := FALSE;
         // apply ReferenceDynamics data to internal ReferenceDynamics data
        _referenceDynamics := ReferenceDynamics;
         // reset data changed bit
         AxesGroup.State.DataChanged.ReferenceDynamics := FALSE;
         // set timeout
         SetTimeout(PT := _rTimeout, rTimer := _rTimer);
         // dec step counter
        _rStep := _rStep - 2;
       ELSE
         // check error ?
         IF (_writeRobotReferenceDynamics.Error)
         THEN
           WarningID := RobotLibraryWarningIdEnum.WARN_REFERENCE_DYNAMICS_SYNC_FAILED_BY_ERROR_OF_READ_OR_WRITE_CMD;
         END_IF

         // timeout exceeded ?
         IF (CheckTimeout(_rTimer) = RobotLibraryConstants.OK)
         THEN
           ErrorID     := RobotLibraryErrorIdEnum.ERR_TIMEOUT_CMD;
           ErrorAddTxt := CONCAT(_stepName, DINT_TO_STRING(_rStep));
         END_IF
       END_IF

    // --------------------------------------------
    // SyncMode after startup :
    // --------------------------------------------

    10 : // check synchronisation active ?
         IF ( AxesGroup.Parameter.Plc.Parameter.SynchronizationModes.ReferenceDynamics[SyncTime.AFTER_START_UP] = SyncMode.NO_SYNCHRONIZATION)
         THEN
           RETURN;
         END_IF

         // compare ReferenceDynamics data
         AxesGroup.State.DataChanged.ReferenceDynamics := NOT IsReferenceDynamicsEqual( Data1 := ReferenceDynamics, Data2 := _referenceDynamics, IgnoreTimestamp := FALSE);

         // Check ReferenceDynamics data changed ?
         IF (AxesGroup.State.DataChanged.ReferenceDynamics)
         THEN
           // Create log entry
           CreateLogMessagePara1 ( Timestamp   := SystemTime,
                                   MessageType := MessageType.CMD,
                                   Severity    := Severity.DEBUG,
                                   MessageCode := 0,
                                   MessageText := 'SyncReferenceDynamics: Detected a local change of ReferenceDynamics on PLC, SyncTime = {1}',
                                   Para1       :=  SYNC_TIME_TO_STRING(SyncTime.AFTER_START_UP));
         END_IF

         // Update plc in sync flag
         AxesGroup.State.SyncStatePlc.InSync.ReferenceDynamics := NOT AxesGroup.State.DataChanged.ReferenceDynamics;

         // Check synchronization is needed ?
         IF ( NOT AxesGroup.State.SyncStatePlc.InSync.ReferenceDynamics ) XOR
            ( NOT AxesGroup.State.SyncStateRc .InSync.ReferenceDynamics )
         THEN
           CASE AxesGroup.Parameter.Plc.Parameter.SynchronizationModes.ReferenceDynamics[SyncTime.AFTER_START_UP]
           OF
             // NO_SYNCHRONIZATION
             SyncMode.NO_SYNCHRONIZATION : ; // no further action

             // CLIENT_TO_SERVER
             SyncMode.CLIENT_TO_SERVER :
               // set timeout
               SetTimeout(PT := _rTimeout, rTimer := _rTimer);
               // inc step counter
              _rStep := 11;

             // SERVER_TO_CLIENT
             SyncMode.SERVER_TO_CLIENT :
               // set timeout
               SetTimeout(PT := _rTimeout, rTimer := _rTimer);
               // inc step counter
              _rStep := 12;

             // AUTOMATIC
             SyncMode.AUTOMATIC :
               // set timeout
               SetTimeout(PT := _rTimeout, rTimer := _rTimer);
               // inc step counter
              _rStep := 13;
           END_CASE
         ELSE
           // datas changeḍ on both sides ? -> Warning
           IF (( NOT AxesGroup.State.SyncStatePlc.InSync.ReferenceDynamics ) AND
               ( NOT AxesGroup.State.SyncStateRc .InSync.ReferenceDynamics ))
           THEN
             WarningID := RobotLibraryWarningIdEnum.WARN_REFERENCE_DYNAMICS_SYNC_BOTH_SIDES_CHANGED;
           END_IF
         END_IF

    // ------------------------------------------
    // SyncMode : CLIENT_TO_SERVER
    // ------------------------------------------
    11 : // Conflict triggerd by PLC ?
         IF ( NOT AxesGroup.State.SyncStatePlc.InSync.ReferenceDynamics )
         THEN
           // set timeout
           SetTimeout(PT := _rTimeout, rTimer := _rTimer);
           // inc step counter
          _rStep := 30; // -> write PLC data to RC

           // Create log entry
           CreateLogMessagePara2 ( Timestamp   := SystemTime,
                                   MessageType := MessageType.CMD,
                                   Severity    := Severity.DEBUG,
                                   MessageCode := 0,
                                   MessageText := 'SyncReferenceDynamics: Synchronization of ReferenceDynamics triggered by PLC, SyncMode = {1}, SyncTime = {2}, SyncDirection = PLC -> RC',
                                   Para1       :=  SYNC_MODE_TO_STRING(AxesGroup.Parameter.Plc.Parameter.SynchronizationModes.ReferenceDynamics[SyncTime.AFTER_START_UP]),
                                   Para2       :=  SYNC_TIME_TO_STRING(SyncTime.AFTER_START_UP));
                                   RETURN;
         END_IF

         // Conflict triggered by RC ?
         IF ( NOT AxesGroup.State.SyncStateRc.InSync.ReferenceDynamics )
         THEN
           // set timeout
           SetTimeout(PT := _rTimeout, rTimer := _rTimer);
           // inc step counter
          _rStep := 30; // -> write PLC data to RC

           // Create log entry
           CreateLogMessagePara2 ( Timestamp   := SystemTime,
                                   MessageType := MessageType.CMD,
                                   Severity    := Severity.DEBUG,
                                   MessageCode := 0,
                                   MessageText := 'SyncReferenceDynamics: Synchronization of ReferenceDynamics triggered by RC, SyncMode = {1}, SyncTime = {2}, SyncDirection = PLC -> RC',
                                   Para1       :=  SYNC_MODE_TO_STRING(AxesGroup.Parameter.Plc.Parameter.SynchronizationModes.ReferenceDynamics[SyncTime.AFTER_START_UP]),
                                   Para2       :=  SYNC_TIME_TO_STRING(SyncTime.AFTER_START_UP));
                                   RETURN;
  			 END_IF

         // set timeout
         SetTimeout(PT := _rTimeout, rTimer := _rTimer);
         // jump back
        _rStep := 10;

    // ------------------------------------------
    // SyncMode : SERVER_TO_CLIENT
    // ------------------------------------------
    12 : // Conflict triggerd by PLC ?
         IF ( NOT AxesGroup.State.SyncStatePlc.InSync.ReferenceDynamics )
         THEN
           // set timeout
           SetTimeout(PT := _rTimeout, rTimer := _rTimer);
           // inc step counter
          _rStep := 20; // -> read RC data and write it to PLC

           // Create log entry
           CreateLogMessagePara2 ( Timestamp   := SystemTime,
                                   MessageType := MessageType.CMD,
                                   Severity    := Severity.DEBUG,
                                   MessageCode := 0,
                                   MessageText := 'SyncReferenceDynamics: Synchronization of ReferenceDynamics triggered by PLC, SyncMode = {1}, SyncTime = {2}, SyncDirection = RC -> PLC',
                                   Para1       :=  SYNC_MODE_TO_STRING(AxesGroup.Parameter.Plc.Parameter.SynchronizationModes.ReferenceDynamics[SyncTime.AFTER_START_UP]),
                                   Para2       :=  SYNC_TIME_TO_STRING(SyncTime.AFTER_START_UP));
                                   RETURN;
         END_IF

         // Conflict triggered by RC ?
         IF ( NOT AxesGroup.State.SyncStateRc.InSync.ReferenceDynamics )
         THEN
           // set timeout
           SetTimeout(PT := _rTimeout, rTimer := _rTimer);
           // inc step counter
          _rStep := 20; // -> read RC data and write it to PLC

           // Create log entry
           CreateLogMessagePara2 ( Timestamp   := SystemTime,
                                   MessageType := MessageType.CMD,
                                   Severity    := Severity.DEBUG,
                                   MessageCode := 0,
                                   MessageText := 'SyncReferenceDynamics: Synchronization of ReferenceDynamics triggered by RC, SyncMode = {1}, SyncTime = {2}, SyncDirection = RC -> PLC',
                                   Para1       :=  SYNC_MODE_TO_STRING(AxesGroup.Parameter.Plc.Parameter.SynchronizationModes.ReferenceDynamics[SyncTime.AFTER_START_UP]),
                                   Para2       :=  SYNC_TIME_TO_STRING(SyncTime.AFTER_START_UP));
                                   RETURN;
  			 END_IF

         // set timeout
         SetTimeout(PT := _rTimeout, rTimer := _rTimer);
         // jump back
        _rStep := 10;

    // ------------------------------------------
    // SyncMode : AUTOMATIC
    // ------------------------------------------
    13 : // Conflict triggerd by PLC ?
         IF ( NOT AxesGroup.State.SyncStatePlc.InSync.ReferenceDynamics )
         THEN
           // set timeout
           SetTimeout(PT := _rTimeout, rTimer := _rTimer);
           // inc step counter
          _rStep := 30; // -> write PLC data to RC

           // Create log entry
           CreateLogMessagePara2 ( Timestamp   := SystemTime,
                                   MessageType := MessageType.CMD,
                                   Severity    := Severity.DEBUG,
                                   MessageCode := 0,
                                   MessageText := 'SyncReferenceDynamics: Synchronization of ReferenceDynamics triggered by PLC, SyncMode = {1}, SyncTime = {2}, SyncDirection = PLC -> RC',
                                   Para1       :=  SYNC_MODE_TO_STRING(AxesGroup.Parameter.Plc.Parameter.SynchronizationModes.ReferenceDynamics[SyncTime.AFTER_START_UP]),
                                   Para2       :=  SYNC_TIME_TO_STRING(SyncTime.AFTER_START_UP));
                                   RETURN;
         END_IF

         // Conflict triggered by RC ?
         IF ( NOT AxesGroup.State.SyncStateRc.InSync.ReferenceDynamics )
         THEN
           // set timeout
           SetTimeout(PT := _rTimeout, rTimer := _rTimer);
           // inc step counter
          _rStep := 20; // -> read RC data an write it to PLC

           // Create log entry
           CreateLogMessagePara2 ( Timestamp   := SystemTime,
                                   MessageType := MessageType.CMD,
                                   Severity    := Severity.DEBUG,
                                   MessageCode := 0,
                                   MessageText := 'SyncReferenceDynamics: Synchronization of ReferenceDynamics triggered by RC, SyncMode = {1}, SyncTime = {2}, SyncDirection = RC -> PLC',
                                   Para1       :=  SYNC_MODE_TO_STRING(AxesGroup.Parameter.Plc.Parameter.SynchronizationModes.ReferenceDynamics[SyncTime.AFTER_START_UP]),
                                   Para2       :=  SYNC_TIME_TO_STRING(SyncTime.AFTER_START_UP));
                                   RETURN;
  			 END_IF

         // set timeout
         SetTimeout(PT := _rTimeout, rTimer := _rTimer);
         // jump back
        //_rStep := 10;

    // ------------------------------------------
    // Read Data from RC and write it to PLC
    // ------------------------------------------
    20 : IF (( NOT _readRobotReferenceDynamics.Busy  ) AND
             ( NOT _readRobotReferenceDynamics.Error ))
         THEN
           // execute command
          _readRobotReferenceDynamics.Execute := TRUE;
           // set timeout
           SetTimeout(PT := _rTimeout, rTimer := _rTimer);
           // inc step counter
          _rStep := _rStep + 1;
         ELSE
           // check error ?
           IF (_readRobotReferenceDynamics.Error)
           THEN
             ErrorID     := _readRobotReferenceDynamics.ErrorID;
             ErrorAddTxt := _readRobotReferenceDynamics.ErrorAddTxt;
           END_IF

           // timeout exceeded ?
           IF (CheckTimeout(_rTimer) = RobotLibraryConstants.OK)
           THEN
             ErrorID     := RobotLibraryErrorIdEnum.ERR_TIMEOUT_CMD;
             ErrorAddTxt := CONCAT(_stepName, DINT_TO_STRING(_rStep));
           END_IF
         END_IF

    21 : IF (( NOT _readRobotReferenceDynamics.Busy  ) AND
             ( NOT _readRobotReferenceDynamics.Error ) AND
             (     _readRobotReferenceDynamics.Done  ))
         THEN
           // reset execution
          _readRobotReferenceDynamics.Execute := FALSE;
           // update internal ReferenceDynamics data
           ReferenceDynamics := _readRobotReferenceDynamics.OutCmd.DynamicValues;
          _referenceDynamics := _readRobotReferenceDynamics.OutCmd.DynamicValues;
           // set timeout
           SetTimeout(PT := _rTimeout, rTimer := _rTimer);
           // inc step counter
          _rStep := 10; // -> jump to after startup
         ELSE
           // check error ?
           IF (_readRobotReferenceDynamics.Error)
           THEN
             ErrorID     := _readRobotReferenceDynamics.ErrorID;
             ErrorAddTxt := _readRobotReferenceDynamics.ErrorAddTxt;
           END_IF

           // timeout exceeded ?
           IF (CheckTimeout(_rTimer) = RobotLibraryConstants.OK)
           THEN
             ErrorID     := RobotLibraryErrorIdEnum.ERR_TIMEOUT_CMD;
             ErrorAddTxt := CONCAT(_stepName, DINT_TO_STRING(_rStep));
           END_IF
         END_IF

    // ------------------------------------------
    // Write data from PLC to RC
    // ------------------------------------------
    30 : IF (( NOT _writeRobotReferenceDynamics.Busy  ) AND
             ( NOT _writeRobotReferenceDynamics.Error ))
         THEN
           // set command parameter
          _writeRobotReferenceDynamics.ParCmd.DynamicValues :=  ReferenceDynamics;
           // execute command
          _writeRobotReferenceDynamics.Execute := TRUE;
           // set timeout
           SetTimeout(PT := _rTimeout, rTimer := _rTimer);
           // inc step counter
          _rStep := _rStep + 1;
         ELSE
           // check error ?
           IF (_writeRobotReferenceDynamics.Error)
           THEN
             ErrorID     := _writeRobotReferenceDynamics.ErrorID;
             ErrorAddTxt := _writeRobotReferenceDynamics.ErrorAddTxt;;
           END_IF

           // timeout exceeded ?
           IF (CheckTimeout(_rTimer) = RobotLibraryConstants.OK)
           THEN
             ErrorID     := RobotLibraryErrorIdEnum.ERR_TIMEOUT_CMD;
             ErrorAddTxt := CONCAT(_stepName, DINT_TO_STRING(_rStep));
           END_IF
         END_IF

    31 : IF (( NOT _writeRobotReferenceDynamics.Busy  ) AND
             ( NOT _writeRobotReferenceDynamics.Error ) AND
             (     _writeRobotReferenceDynamics.Done  ))
         THEN
           // execute command
          _writeRobotReferenceDynamics.Execute := FALSE;
           // update internal ReferenceDynamics data
          _ReferenceDynamics := ReferenceDynamics;
           // set timeout
           SetTimeout(PT := _rTimeout, rTimer := _rTimer);
           // inc step counter
          _rStep := 10; // -> jump to after startup;
         ELSE
           // check error ?
           IF (_writeRobotReferenceDynamics.Error)
           THEN
             WarningID := RobotLibraryWarningIdEnum.WARN_REFERENCE_DYNAMICS_SYNC_FAILED_BY_ERROR_OF_READ_OR_WRITE_CMD;
           END_IF

           // timeout exceeded ?
           IF (CheckTimeout(_rTimer) = RobotLibraryConstants.OK)
           THEN
             ErrorID     := RobotLibraryErrorIdEnum.ERR_TIMEOUT_CMD;
             ErrorAddTxt := CONCAT(_stepName, DINT_TO_STRING(_rStep));
           END_IF
         END_IF

  ELSE
    // invalid step
    ErrorID     := RobotLibraryErrorIdEnum.ERR_INVALID_STEP;
    ErrorAddTxt := CONCAT(_stepName , DINT_TO_STRING(_stepCmd));
  END_CASE

END_METHOD

METHOD PRIVATE HandleSyncRobotSWLimits
VAR_IN_OUT
   /// Robot assignment of function
  AxesGroup : AxesGroup;
  /// Software limits stored on PLC
  SWLimits  : SWLimits;
END_VAR

VAR
  /// Internal step counter name
 _stepName        : STRING;
  /// Internal reference to step counter
 _rStep           : REFERENCE TO DINT;
  /// Internal reference to timer
 _rTimer          : REFERENCE TO TON;
  /// Internal reference to timeout
 _rTimeout        : REFERENCE TO TIME;
  /// empty data set to reset all DataChanged bits
 _dataChangedNone : AxesGroupStateDataChanged;
END_VAR

  // Set internal references
  _stepName      :=   '_stepSyncSWLimits = ';
  _rStep       REF=    _stepSyncSWLimits;
  _rTimer      REF=   _timerSyncSWLimits;
  _rTimeout    REF= _timeoutSyncSWLimits;

  CASE _rStep
  OF
    0: // Check initialisation configured ?
       IF (( _parCfg.PLC.Parameter.SynchronizationModes.SWLimits[SyncTime.DURING_START_UP] = SyncMode.NO_SYNCHRONIZATION ) AND
           ( _parCfg.PLC.Parameter.SynchronizationModes.SWLimits[SyncTime. AFTER_START_UP] = SyncMode.NO_SYNCHRONIZATION ))
       THEN
         RETURN;
       END_IF

       // wait for initialisation done
       IF  ((     AxesGroup.State.RobotData.RCSupportedFunctions .ReadRobotSWLimits ) AND
            (     AxesGroup.State.RobotData.RCSupportedFunctions.WriteRobotSWLimits ) AND
            (     AxesGroup.State.Initialized                                       ) AND
            ( NOT Error                                                             ))
       THEN
         // Create log entry
         CreateLogMessagePara1 ( Timestamp   := SystemTime,
                                 MessageType := MessageType.CMD,
                                 Severity    := Severity.DEBUG,
                                 MessageCode := 0,
                                 MessageText := 'SyncSwLimits: Start initial reading of SwLimits from RC',
                                 Para1       :=  '');

         // set timeout
         SetTimeout(PT := _rTimeout, rTimer := _rTimer);
         // inc step counter
        _rStep := _rStep + 1;
       END_IF

       // Start read SwLimits
    1: IF (( NOT _readRobotSWLimits .Busy  ) AND
           ( NOT _readRobotSWLimits.Error ))
       THEN
         // execute command
        _readRobotSWLimits.Execute := TRUE;
         // set timeout
         SetTimeout(PT := _rTimeout, rTimer := _rTimer);
         // inc step counter
        _rStep := _rStep + 1;
       ELSE
         // check error ?
         IF ( _readRobotSWLimits.Error ) AND ( WarningID = RobotLibraryWarningIdEnum.NO_WARNING )
         THEN
           WarningID := RobotLibraryWarningIdEnum.WARN_SW_LIMITS_SYNC_FAILED_BY_ERROR_OF_READ_OR_WRITE_CMD;
         END_IF

         // timeout exceeded ?
         IF (CheckTimeout(_rTimer) = RobotLibraryConstants.OK)
         THEN
           ErrorID     := RobotLibraryErrorIdEnum.ERR_TIMEOUT_CMD;
           ErrorAddTxt := CONCAT(_stepName, DINT_TO_STRING(_rStep));
         END_IF
       END_IF

       // Wait SwLimits read
    2: IF (( NOT _readRobotSWLimits.Busy  ) AND
           ( NOT _readRobotSWLimits.Error ) AND
           (     _readRobotSWLimits.Done  ))
       THEN
         // reset execution
        _readRobotSWLimits.Execute := FALSE;
         // Copy data
        _swLimits := _readRobotSWLimits.OutCmd.LimitValues;
         // Set plc in sync flag
         AxesGroup.State.SyncStatePlc.InSync.SwLimits := TRUE;

         // Check SwLimits data is equal ?
         IF ( NOT IsSwLimitsEqual( Data1 := _swLimits, Data2 := SwLimits, IgnoreTimestamp := TRUE))
         THEN
           // Reset plc in sync flag
           AxesGroup.State.SyncStatePlc.InSync.SwLimits := FALSE;
           // Set data changed flag
           AxesGroup.State.DataChanged.SwLimits := TRUE;
           // set timeout
           SetTimeout(PT := _rTimeout, rTimer := _rTimer);
           // inc step counter
          _rStep := _rStep + 1;

           // Create log entry
           CreateLogMessagePara1 ( Timestamp   := SystemTime,
                                   MessageType := MessageType.CMD,
                                   Severity    := Severity.DEBUG,
                                   MessageCode := 0,
                                   MessageText := 'SyncSwLimits: Detected a difference in SwLimits between PLC and RC',
                                   Para1       :=  '');

           // Check synchronisation is enabled ?
           IF ( NOT  AxesGroup.State.DataEnableSync.EnableSyncSWLimits ) AND (InfoID = RobotLibraryInfoIdEnum.NO_INFO )
           THEN
             InfoID := RobotLibraryInfoIdEnum.INFO_SYNC_SWLIMIT_DISABLED;
  				 END_IF

           // Check user interaction needed ?
           IF ( AxesGroup.Parameter.Plc.Parameter.SyncUserInteraction.SWLimits ) AND ( WarningID = RobotLibraryWarningIdEnum.NO_WARNING )
           THEN
             WarningID := RobotLibraryWarningIdEnum.WARN_SW_LIMITS_SYNC_ERROR;
  				 END_IF
  			 END_IF
       ELSE
         // check error ?
         IF (_readRobotSWLimits.Error)
         THEN
           // Set warning
           WarningID := RobotLibraryWarningIdEnum.WARN_SW_LIMITS_SYNC_FAILED_BY_ERROR_OF_READ_OR_WRITE_CMD;
         END_IF

         // timeout exceeded ?
         IF (CheckTimeout(_rTimer) = RobotLibraryConstants.OK)
         THEN
           ErrorID     := RobotLibraryErrorIdEnum.ERR_TIMEOUT_CMD;
           ErrorAddTxt := CONCAT(_stepName, DINT_TO_STRING(_rStep));
         END_IF
       END_IF

       // Check synchronisation state ?
    3: IF ((  NOT AxesGroup.State.DataChanged.SwLimits                                                                                    ) OR
           (      AxesGroup.Parameter.Plc.Parameter.SynchronizationModes.SWLimits[SyncTime.DURING_START_UP] = SyncMode.NO_SYNCHRONIZATION ))
       THEN
         // Update bit for data in sync
         AxesGroup.State.SyncStatePlc.InSync.SwLimits := NOT AxesGroup.State.DataChanged.SwLimits ;
         // set timeout
         SetTimeout(PT := _rTimeout, rTimer := _rTimer);
         // inc step counter
        _rStep := 10; // -> jump to after startup

         // Create log entry
         CreateLogMessagePara1 ( Timestamp   := SystemTime,
                                 MessageType := MessageType.CMD,
                                 Severity    := Severity.DEBUG,
                                 MessageCode := 0,
                                 MessageText := 'SyncSwLimits: Synchronization Startup Phase done',
                                 Para1       :=  '' );
       ELSE
         // Check user interaction needed ?
         IF ( NOT AxesGroup.Parameter.Plc.Parameter.SyncUserInteraction.SWLimits )
         THEN
           CASE AxesGroup.Parameter.Plc.Parameter.SynchronizationModes.SWLimits[SyncTime.DURING_START_UP] OF

             SyncMode.SERVER_TO_CLIENT :

               // Overwrite PLC data with RC data
               SwLimits := _swLimits;
               // Reset data changed flags
               AxesGroup.State.DataChanged.SwLimits := _dataChangedNone.SwLimits;
               // Reset Synchronizing flag
               AxesGroup.State.Synchronizing.SwLimits := FALSE;
               // Set plc in sync flag
               AxesGroup.State.SyncStatePlc.InSync.SwLimits := TRUE;
               // set timeout
               SetTimeout(PT := _rTimeout, rTimer := _rTimer);
               // inc step counter
              _rStep := 10; // -> jump to after startup

              // Create log entry
              CreateLogMessagePara2 ( Timestamp   := SystemTime,
                                      MessageType := MessageType.CMD,
                                      Severity    := Severity.DEBUG,
                                      MessageCode := 0,
                                      MessageText := 'SyncSwLimits: Synchronization of SwLimits triggered by StartUp-Compare, SyncMode = {1}, SyncTime = {2}, SyncDirection = RC -> PLC',
                                      Para1       :=  SYNC_MODE_TO_STRING(AxesGroup.Parameter.Plc.Parameter.SynchronizationModes.SWLimits[SyncTime.DURING_START_UP]),
                                      Para2       :=  SYNC_TIME_TO_STRING(SyncTime.DURING_START_UP));
              // Create log entry
              CreateLogMessagePara1 ( Timestamp   := SystemTime,
                                      MessageType := MessageType.CMD,
                                      Severity    := Severity.DEBUG,
                                      MessageCode := 0,
                                      MessageText := 'SyncSwLimits: Applied the initial read SwLimits from RC',
                                      Para1       :=  '' );

  				   SyncMode.CLIENT_TO_SERVER : ;

               IF ( AxesGroup.State.DataChanged.SwLimits )
               THEN
                 // Reset plc in sync flag
                 AxesGroup.State.SyncStatePlc.InSync.SwLimits := FALSE;
                 // Set Synchronizing flag
                 AxesGroup.State.Synchronizing.SwLimits := TRUE;
                 // set timeout
                 SetTimeout(PT := _rTimeout, rTimer := _rTimer);
                 // inc step counter
                _rStep := _rStep +1; // -> write PLC data to RC
                 // Create log entry
                 CreateLogMessagePara2 ( Timestamp   := SystemTime,
                                         MessageType := MessageType.CMD,
                                         Severity    := Severity.DEBUG,
                                         MessageCode := 0,
                                         MessageText := 'SyncSwLimits: Synchronization of SwLimits triggered by StartUp-Compare, SyncMode = {1}, SyncTime = {2}, SyncDirection = PLC -> RC',
                                         Para1       :=  SYNC_MODE_TO_STRING(AxesGroup.Parameter.Plc.Parameter.SynchronizationModes.SWLimits[SyncTime.DURING_START_UP]),
                                         Para2       :=  SYNC_TIME_TO_STRING(SyncTime.DURING_START_UP));
               ELSE
                 // Reset data changed flags
                 AxesGroup.State.DataChanged.SwLimits := _dataChangedNone.SwLimits;
                 // Reset Synchronizing flag
                 AxesGroup.State.Synchronizing.SwLimits := FALSE;
                 // Set plc in sync flag
                 AxesGroup.State.SyncStatePlc.InSync.SwLimits := TRUE;
                 // set timeout
                 SetTimeout(PT := _rTimeout, rTimer := _rTimer);
                 // inc step counter
                _rStep := 10; // -> jump to after startup
  				     END_IF
           ELSE
             // invalid sync mode for startup
             ErrorID := RobotLibraryErrorIdEnum.ERR_SYNC_MODE_INVALID;
   	       END_CASE
         END_IF
       END_IF

       // Start write SwLimits data
    4: IF (( NOT _writeRobotSWLimits.Busy  ) AND
           ( NOT _writeRobotSWLimits.Error ))
       THEN
         // set command parameter
        _writeRobotSWLimits.ParCmd.LimitValues :=  SwLimits;
        _writeRobotSWLimits.ParCmd.ResetToFactoryDefaults := FALSE;
         // execute command
        _writeRobotSWLimits.Execute := TRUE;
         // set timeout
         SetTimeout(PT := _rTimeout, rTimer := _rTimer);
         // inc step counter
        _rStep := _rStep + 1;
       ELSE
         // check error ?
         IF (_writeRobotSWLimits.Error)
         THEN
           ErrorID     := _writeRobotSWLimits.ErrorID;
           ErrorAddTxt := _writeRobotSWLimits.ErrorAddTxt;;
         END_IF

         // timeout exceeded ?
         IF (CheckTimeout(_rTimer) = RobotLibraryConstants.OK)
         THEN
           ErrorID     := RobotLibraryErrorIdEnum.ERR_TIMEOUT_CMD;
           ErrorAddTxt := CONCAT(_stepName, DINT_TO_STRING(_rStep));
         END_IF
       END_IF

       // Wait SwLimits data written ?
    5: IF (( NOT _writeRobotSWLimits.Busy  ) AND
           ( NOT _writeRobotSWLimits.Error ) AND
           (     _writeRobotSWLimits.Done  ))
       THEN
         // execute command
        _writeRobotSWLimits.Execute := FALSE;
         // apply SwLimits data to internal SwLimits data
        _swLimits := SwLimits;
         // reset data changed bit
         AxesGroup.State.DataChanged.SwLimits := FALSE;
         // set timeout
         SetTimeout(PT := _rTimeout, rTimer := _rTimer);
         // dec step counter
        _rStep := _rStep - 2;
       ELSE
         // check error ?
         IF (_writeRobotSWLimits.Error)
         THEN
           WarningID := RobotLibraryWarningIdEnum.WARN_SW_LIMITS_SYNC_FAILED_BY_ERROR_OF_READ_OR_WRITE_CMD;
         END_IF

         // timeout exceeded ?
         IF (CheckTimeout(_rTimer) = RobotLibraryConstants.OK)
         THEN
           ErrorID     := RobotLibraryErrorIdEnum.ERR_TIMEOUT_CMD;
           ErrorAddTxt := CONCAT(_stepName, DINT_TO_STRING(_rStep));
         END_IF
       END_IF

    // --------------------------------------------
    // SyncMode after startup :
    // --------------------------------------------

    10 : // check synchronisation active ?
         IF ( AxesGroup.Parameter.Plc.Parameter.SynchronizationModes.SWLimits[SyncTime.AFTER_START_UP] = SyncMode.NO_SYNCHRONIZATION)
         THEN
           RETURN;
         END_IF

         // compare SwLimits data
         AxesGroup.State.DataChanged.SwLimits := NOT IsSwLimitsEqual( Data1 := SwLimits, Data2 := _swLimits, IgnoreTimestamp := FALSE);

         // Check SwLimits data changed ?
         IF (AxesGroup.State.DataChanged.SwLimits)
         THEN
           // Create log entry
           CreateLogMessagePara1 ( Timestamp   := SystemTime,
                                   MessageType := MessageType.CMD,
                                   Severity    := Severity.DEBUG,
                                   MessageCode := 0,
                                   MessageText := 'SyncSwLimits: Detected a local change of SwLimits on PLC, SyncTime = {1}',
                                   Para1       :=  SYNC_TIME_TO_STRING(SyncTime.AFTER_START_UP));
         END_IF

         // Update plc in sync flag
         AxesGroup.State.SyncStatePlc.InSync.SwLimits := NOT AxesGroup.State.DataChanged.SwLimits;

         // Check synchronization is needed ?
         IF ( NOT AxesGroup.State.SyncStatePlc.InSync.SwLimits ) XOR
            ( NOT AxesGroup.State.SyncStateRc .InSync.SwLimits )
         THEN
           CASE AxesGroup.Parameter.Plc.Parameter.SynchronizationModes.SWLimits[SyncTime.AFTER_START_UP]
           OF
             // NO_SYNCHRONIZATION
             SyncMode.NO_SYNCHRONIZATION : ; // no further action

             // CLIENT_TO_SERVER
             SyncMode.CLIENT_TO_SERVER :
               // set timeout
               SetTimeout(PT := _rTimeout, rTimer := _rTimer);
               // inc step counter
              _rStep := 11;

             // SERVER_TO_CLIENT
             SyncMode.SERVER_TO_CLIENT :
               // set timeout
               SetTimeout(PT := _rTimeout, rTimer := _rTimer);
               // inc step counter
              _rStep := 12;

             // AUTOMATIC
             SyncMode.AUTOMATIC :
               // set timeout
               SetTimeout(PT := _rTimeout, rTimer := _rTimer);
               // inc step counter
              _rStep := 13;
           END_CASE
         ELSE
           // datas changeḍ on both sides ? -> Warning
           IF (( NOT AxesGroup.State.SyncStatePlc.InSync.SwLimits ) AND
               ( NOT AxesGroup.State.SyncStateRc .InSync.SwLimits ))
           THEN
             WarningID := RobotLibraryWarningIdEnum.WARN_SW_LIMITS_SYNC_BOTH_SIDES_CHANGED;
           END_IF
         END_IF

    // ------------------------------------------
    // SyncMode : CLIENT_TO_SERVER
    // ------------------------------------------
    11 : // Conflict triggerd by PLC ?
         IF ( NOT AxesGroup.State.SyncStatePlc.InSync.SwLimits )
         THEN
           // set timeout
           SetTimeout(PT := _rTimeout, rTimer := _rTimer);
           // inc step counter
          _rStep := 30; // -> write PLC data to RC

           // Create log entry
           CreateLogMessagePara2 ( Timestamp   := SystemTime,
                                   MessageType := MessageType.CMD,
                                   Severity    := Severity.DEBUG,
                                   MessageCode := 0,
                                   MessageText := 'SyncSwLimits: Synchronization of SwLimits triggered by PLC, SyncMode = {1}, SyncTime = {2}, SyncDirection = PLC -> RC',
                                   Para1       :=  SYNC_MODE_TO_STRING(AxesGroup.Parameter.Plc.Parameter.SynchronizationModes.SWLimits[SyncTime.AFTER_START_UP]),
                                   Para2       :=  SYNC_TIME_TO_STRING(SyncTime.AFTER_START_UP));
                                   RETURN;
         END_IF

         // Conflict triggered by RC ?
         IF ( NOT AxesGroup.State.SyncStateRc.InSync.SwLimits )
         THEN
           // set timeout
           SetTimeout(PT := _rTimeout, rTimer := _rTimer);
           // inc step counter
          _rStep := 30; // -> write PLC data to RC

           // Create log entry
           CreateLogMessagePara2 ( Timestamp   := SystemTime,
                                   MessageType := MessageType.CMD,
                                   Severity    := Severity.DEBUG,
                                   MessageCode := 0,
                                   MessageText := 'SyncSwLimits: Synchronization of SwLimits triggered by RC, SyncMode = {1}, SyncTime = {2}, SyncDirection = PLC -> RC',
                                   Para1       :=  SYNC_MODE_TO_STRING(AxesGroup.Parameter.Plc.Parameter.SynchronizationModes.SWLimits[SyncTime.AFTER_START_UP]),
                                   Para2       :=  SYNC_TIME_TO_STRING(SyncTime.AFTER_START_UP));
                                   RETURN;
  			 END_IF

         // set timeout
         SetTimeout(PT := _rTimeout, rTimer := _rTimer);
         // jump back
        _rStep := 10;

    // ------------------------------------------
    // SyncMode : SERVER_TO_CLIENT
    // ------------------------------------------
    12 : // Conflict triggerd by PLC ?
         IF ( NOT AxesGroup.State.SyncStatePlc.InSync.SwLimits )
         THEN
           // set timeout
           SetTimeout(PT := _rTimeout, rTimer := _rTimer);
           // inc step counter
          _rStep := 20; // -> read RC data and write it to PLC

           // Create log entry
           CreateLogMessagePara2 ( Timestamp   := SystemTime,
                                   MessageType := MessageType.CMD,
                                   Severity    := Severity.DEBUG,
                                   MessageCode := 0,
                                   MessageText := 'SyncSwLimits: Synchronization of SwLimits triggered by PLC, SyncMode = {1}, SyncTime = {2}, SyncDirection = RC -> PLC',
                                   Para1       :=  SYNC_MODE_TO_STRING(AxesGroup.Parameter.Plc.Parameter.SynchronizationModes.SWLimits[SyncTime.AFTER_START_UP]),
                                   Para2       :=  SYNC_TIME_TO_STRING(SyncTime.AFTER_START_UP));
                                   RETURN;
         END_IF

         // Conflict triggered by RC ?
         IF ( NOT AxesGroup.State.SyncStateRc.InSync.SwLimits )
         THEN
           // set timeout
           SetTimeout(PT := _rTimeout, rTimer := _rTimer);
           // inc step counter
          _rStep := 20; // -> read RC data and write it to PLC

           // Create log entry
           CreateLogMessagePara2 ( Timestamp   := SystemTime,
                                   MessageType := MessageType.CMD,
                                   Severity    := Severity.DEBUG,
                                   MessageCode := 0,
                                   MessageText := 'SyncSwLimits: Synchronization of SwLimits triggered by RC, SyncMode = {1}, SyncTime = {2}, SyncDirection = RC -> PLC',
                                   Para1       :=  SYNC_MODE_TO_STRING(AxesGroup.Parameter.Plc.Parameter.SynchronizationModes.SWLimits[SyncTime.AFTER_START_UP]),
                                   Para2       :=  SYNC_TIME_TO_STRING(SyncTime.AFTER_START_UP));
                                   RETURN;
  			 END_IF

         // set timeout
         SetTimeout(PT := _rTimeout, rTimer := _rTimer);
         // jump back
        _rStep := 10;

    // ------------------------------------------
    // SyncMode : AUTOMATIC
    // ------------------------------------------
    13 : // Conflict triggerd by PLC ?
         IF ( NOT AxesGroup.State.SyncStatePlc.InSync.SwLimits )
         THEN
           // set timeout
           SetTimeout(PT := _rTimeout, rTimer := _rTimer);
           // inc step counter
          _rStep := 30; // -> write PLC data to RC

           // Create log entry
           CreateLogMessagePara2 ( Timestamp   := SystemTime,
                                   MessageType := MessageType.CMD,
                                   Severity    := Severity.DEBUG,
                                   MessageCode := 0,
                                   MessageText := 'SyncSwLimits: Synchronization of SwLimits triggered by PLC, SyncMode = {1}, SyncTime = {2}, SyncDirection = PLC -> RC',
                                   Para1       :=  SYNC_MODE_TO_STRING(AxesGroup.Parameter.Plc.Parameter.SynchronizationModes.SWLimits[SyncTime.AFTER_START_UP]),
                                   Para2       :=  SYNC_TIME_TO_STRING(SyncTime.AFTER_START_UP));
                                   RETURN;
         END_IF

         // Conflict triggered by RC ?
         IF ( NOT AxesGroup.State.SyncStateRc.InSync.SwLimits )
         THEN
           // set timeout
           SetTimeout(PT := _rTimeout, rTimer := _rTimer);
           // inc step counter
          _rStep := 20; // -> read RC data an write it to PLC

           // Create log entry
           CreateLogMessagePara2 ( Timestamp   := SystemTime,
                                   MessageType := MessageType.CMD,
                                   Severity    := Severity.DEBUG,
                                   MessageCode := 0,
                                   MessageText := 'SyncSwLimits: Synchronization of SwLimits triggered by RC, SyncMode = {1}, SyncTime = {2}, SyncDirection = RC -> PLC',
                                   Para1       :=  SYNC_MODE_TO_STRING(AxesGroup.Parameter.Plc.Parameter.SynchronizationModes.SWLimits[SyncTime.AFTER_START_UP]),
                                   Para2       :=  SYNC_TIME_TO_STRING(SyncTime.AFTER_START_UP));
                                   RETURN;
  			 END_IF

         // set timeout
         SetTimeout(PT := _rTimeout, rTimer := _rTimer);
         // jump back
        //_rStep := 10;

    // ------------------------------------------
    // Read Data from RC and write it to PLC
    // ------------------------------------------
    20 : IF (( NOT _readRobotSWLimits.Busy  ) AND
             ( NOT _readRobotSWLimits.Error ))
         THEN
           // execute command
          _readRobotSWLimits.Execute := TRUE;
           // set timeout
           SetTimeout(PT := _rTimeout, rTimer := _rTimer);
           // inc step counter
          _rStep := _rStep + 1;
         ELSE
           // check error ?
           IF (_readRobotSWLimits.Error)
           THEN
             ErrorID     := _readRobotSWLimits.ErrorID;
             ErrorAddTxt := _readRobotSWLimits.ErrorAddTxt;
           END_IF

           // timeout exceeded ?
           IF (CheckTimeout(_rTimer) = RobotLibraryConstants.OK)
           THEN
             ErrorID     := RobotLibraryErrorIdEnum.ERR_TIMEOUT_CMD;
             ErrorAddTxt := CONCAT(_stepName, DINT_TO_STRING(_rStep));
           END_IF
         END_IF

    21 : IF (( NOT _readRobotSWLimits.Busy  ) AND
             ( NOT _readRobotSWLimits.Error ) AND
             (     _readRobotSWLimits.Done  ))
         THEN
           // reset execution
          _readRobotSWLimits.Execute := FALSE;
           // update internal SwLimits data
           SwLimits := _readRobotSWLimits.OutCmd.LimitValues;
          _swLimits := _readRobotSWLimits.OutCmd.LimitValues;
           // set timeout
           SetTimeout(PT := _rTimeout, rTimer := _rTimer);
           // inc step counter
          _rStep := 10; // -> jump to after startup
         ELSE
           // check error ?
           IF (_readRobotSWLimits.Error)
           THEN
             ErrorID     := _readRobotSWLimits.ErrorID;
             ErrorAddTxt := _readRobotSWLimits.ErrorAddTxt;
           END_IF

           // timeout exceeded ?
           IF (CheckTimeout(_rTimer) = RobotLibraryConstants.OK)
           THEN
             ErrorID     := RobotLibraryErrorIdEnum.ERR_TIMEOUT_CMD;
             ErrorAddTxt := CONCAT(_stepName, DINT_TO_STRING(_rStep));
           END_IF
         END_IF

    // ------------------------------------------
    // Write data from PLC to RC
    // ------------------------------------------
    30 : IF (( NOT _writeRobotSWLimits.Busy  ) AND
             ( NOT _writeRobotSWLimits.Error ))
         THEN
           // set command parameter
          _writeRobotSWLimits.ParCmd.ResetToFactoryDefaults := FALSE;
          _writeRobotSWLimits.ParCmd.LimitValues :=  SwLimits;
           // execute command
          _writeRobotSWLimits.Execute := TRUE;
           // set timeout
           SetTimeout(PT := _rTimeout, rTimer := _rTimer);
           // inc step counter
          _rStep := _rStep + 1;
         ELSE
           // check error ?
           IF (_writeRobotSWLimits.Error)
           THEN
             ErrorID     := _writeRobotSWLimits.ErrorID;
             ErrorAddTxt := _writeRobotSWLimits.ErrorAddTxt;;
           END_IF

           // timeout exceeded ?
           IF (CheckTimeout(_rTimer) = RobotLibraryConstants.OK)
           THEN
             ErrorID     := RobotLibraryErrorIdEnum.ERR_TIMEOUT_CMD;
             ErrorAddTxt := CONCAT(_stepName, DINT_TO_STRING(_rStep));
           END_IF
         END_IF

    31 : IF (( NOT _writeRobotSWLimits.Busy  ) AND
             ( NOT _writeRobotSWLimits.Error ) AND
             (     _writeRobotSWLimits.Done  ))
         THEN
           // execute command
          _writeRobotSWLimits.Execute := FALSE;
           // update internal SwLimits data
          _swLimits := SwLimits;
           // set timeout
           SetTimeout(PT := _rTimeout, rTimer := _rTimer);
           // inc step counter
          _rStep := 10; // -> jump to after startup;
         ELSE
           // check error ?
           IF (_writeRobotSWLimits.Error)
           THEN
             WarningID := RobotLibraryWarningIdEnum.WARN_SW_LIMITS_SYNC_FAILED_BY_ERROR_OF_READ_OR_WRITE_CMD;
           END_IF

           // timeout exceeded ?
           IF (CheckTimeout(_rTimer) = RobotLibraryConstants.OK)
           THEN
             ErrorID     := RobotLibraryErrorIdEnum.ERR_TIMEOUT_CMD;
             ErrorAddTxt := CONCAT(_stepName, DINT_TO_STRING(_rStep));
           END_IF
         END_IF

  ELSE
    // invalid step
    ErrorID     := RobotLibraryErrorIdEnum.ERR_INVALID_STEP;
    ErrorAddTxt := CONCAT(_stepName , DINT_TO_STRING(_stepCmd));
  END_CASE

END_METHOD

METHOD PRIVATE HandleSyncToolData
VAR_IN_OUT
   /// Robot assignment of function
  AxesGroup : AxesGroup;
  /// ToolData stored on PLC.For more information refer to 5.5.6.4
  ToolData  : ARRAY[0..RobotLibraryParameter.TOOL_MAX -1] OF Tool;
END_VAR

VAR
  /// Internal step counter name
 _stepName        : STRING;
  /// Internal reference to step counter
 _rStep           : REFERENCE TO DINT;
  /// Internal reference to timer
 _rTimer          : REFERENCE TO TON;
  /// Internal reference to timeout
 _rTimeout        : REFERENCE TO TIME;
  /// Internal reference to synchroniztion index
 _rSyncIdx        : REFERENCE TO USINT;
  /// internal bit for condition found
 _found           : BOOL;
  /// empty data set to reset all DataChanged bits
 _dataChangedNone : AxesGroupStateDataChanged;
END_VAR

  // Set internal references
  _stepName      :=   '_stepSyncToolData = ';
  _rStep       REF=    _stepSyncToolData;
  _rTimer      REF=   _timerSyncToolData;
  _rTimeout    REF= _timeoutSyncToolData;
  _rSyncIdx    REF=     _syncIdxToolData;

  CASE _rStep
  OF
    0: // Check initialisation configured ?
       IF (( _parCfg.PLC.Parameter.SynchronizationModes.SWLimits[SyncTime.DURING_START_UP] = SyncMode.NO_SYNCHRONIZATION ) AND
           ( _parCfg.PLC.Parameter.SynchronizationModes.SWLimits[SyncTime. AFTER_START_UP] = SyncMode.NO_SYNCHRONIZATION ))
       THEN
         RETURN;
       END_IF

       // wait for initialisation done
       IF  ((     AxesGroup.State.RobotData.RCSupportedFunctions. ReadToolData ) AND
            (     AxesGroup.State.RobotData.RCSupportedFunctions.WriteToolData ) AND
            (     AxesGroup.State.Initialized                                  ) AND
            ( NOT Error                                                        ))
       THEN
         // Check PLC tools < RC tools and SyncTool enabled ?
         IF (( AxesGroup.State.DataEnableSync.EnableSyncTool      = TRUE                              )  AND
             ( AxesGroup.Parameter.Rob.Parameter.HighestToolIndex > RobotLibraryParameter.Tool_MAX -1 ))
         THEN
           WarningID := RobotLibraryWarningIdEnum.WARN_TOOL_DATA_ARRAY_TOO_SHORT;
         END_IF

         // Create log entry
         CreateLogMessagePara1 ( Timestamp   := SystemTime,
                                 MessageType := MessageType.CMD,
                                 Severity    := Severity.DEBUG,
                                 MessageCode := 0,
                                 MessageText := 'SyncToolData: Start initial reading of ToolData from RC',
                                 Para1       :=  '');

         // init tool number
        _rSyncIdx := 0;
         // init count of unsynchronized elements
         AxesGroup.State.SyncStatePlc.UnSyncNo.Tool := 0;
         // set timeout
         SetTimeout(PT := _rTimeout, rTimer := _rTimer);
         // inc step counter
        _rStep := _rStep + 1;
       END_IF

       // Start read ToolData
    1: IF (( NOT _readToolData.Busy  ) AND
           ( NOT _readToolData.Error ))
       THEN
         // set command parameter
        _readToolData.ParCmd.ToolNo := _rSyncIdx;
         // execute command
        _readToolData.Execute := TRUE;
         // set timeout
         SetTimeout(PT := _rTimeout, rTimer := _rTimer);
         // inc step counter
        _rStep := _rStep + 1;
       ELSE
         // check error ?
         IF ( _readToolData.Error ) AND ( WarningID = RobotLibraryWarningIdEnum.NO_WARNING )
         THEN
           WarningID := RobotLibraryWarningIdEnum.WARN_TOOL_SYNC_FAILED_BY_ERROR_OF_READ_OR_WRITE_CMD;
         END_IF
